//==================================================================================================
//							Beckhoff Automation Poland
//									23.05.2017
//	Program obslugujacy wizualizacje VISU_EventsHistoricalSimple
//	Mozliwe filtrowanie alamow. Czestotliwosc odswiezania wplywa tylko na wyswietlanie
// 	v1.0	|| TC v 3.1.4020.32		|| - pierwsza wersja
//==================================================================================================
PROGRAM P_EventsVisu
VAR
	i										: DINT;				// Iterator tablicy przechowywanej w pamieci
	j										: DINT;				// Iterator tablicy wyswietlanej
	bActiveWindow							: BOOL := TRUE;		// Flaga wysietlania okna - tylko wtedy odswiezamy tablice wyswietlana
	rtPageChange							: R_TRIG;			// Wykrycie przelaczenia strony
	tonRefresh								: TON;
	tRefreshTime							: TIME := T#50MS;	// Czestotliwosc odswiezania strony
	//========================= Filtry =========================
	bRemoveFromList							: BOOL; 			// Flaga pomocnicza dla filtrow - decyduje czy element ma byc dodany na wizualizacje
	// Flagi wykonywalnosci
	bFilterID								: BOOL;
	bFilterClass							: BOOL;
	bFilterActiveOnly						: BOOL;
	// Parametry
	dwFilterID								: DWORD;	
	dwFilterClass							: DWORD;
END_VAR

bActiveWindow := TRUE;//VisuElems.CURRENTVISU = 'VISU_EventsHistoricalSimple';						// Flaga wysietlania okna
rtPageChange(CLK:= bActiveWindow, Q=> );													// Wykrycie zmiany strony - jednorazowo inicjalizacja
tonRefresh(IN:= bActiveWindow AND NOT tonRefresh.Q, PT:= tRefreshTime, Q=> , ET=> );		// Timer odswiezania

IF  rtPageChange.Q OR tonRefresh.Q THEN
	// Czyszczenie tablicy
	MEMSET(ADR(GVL_EHS.arrEventVisu),0,SIZEOF(GVL_EHS.arrEventVisu));
	j := 1;
	// Filters
	FOR i := 1 TO GVL_EHS.diNoOfEvents DO
		bRemoveFromList 								:= FALSE;
		// Jesli jest element
		IF GVL_EHSP.arrEvent[i].dwID <> 0 THEN
			bRemoveFromList								:= bFilterID AND dwFilterID <> GVL_EHSP.arrEvent[i].dwID;
			bRemoveFromList								:= bRemoveFromList OR (bFilterClass AND dwFilterClass <> GVL_EHSP.arrEvent[i].dwClass);
//			bRemoveFromList								:= bRemoveFromList OR (bFilterBeginTimeFrom AND GVL_EHSP.arrEvent[i].dtDateBegin <= dtFilterBeginTimeFrom);
//			bRemoveFromList								:= bRemoveFromList OR (bFilterBeginTimeTo AND GVL_EHSP.arrEvent[i].dtDateBegin >= dtFilterBeginTimeTo);
//			bRemoveFromList								:= bRemoveFromList OR (bFilterEndTimeFrom AND GVL_EHSP.arrEvent[i].dtDateEnd <= dtFilterEndTimeFrom);
//			bRemoveFromList								:= bRemoveFromList OR (bFilterEndTimeTo AND GVL_EHSP.arrEvent[i].dtDateEnd >= dtFilterEndTimeTo);
			bRemoveFromList								:= bRemoveFromList OR (bFilterActiveOnly AND DT#1970-1-1-0:0:0 <> GVL_EHSP.arrEvent[i].dtDateEnd);
			// Analogicznie dodajemy inne filtry jesli jest taka potrzeba
			// Jesli element nie zostal usuniety przez filtr to dodajemy go do tablicy alarmow wyswietlanych
			IF NOT bRemoveFromList THEN
				GVL_EHS.arrEventVisu[j].dwID 			:= GVL_EHSP.arrEvent[i].dwID;
				GVL_EHS.arrEventVisu[j].dwClass 		:= GVL_EHSP.arrEvent[i].dwClass;
				GVL_EHS.arrEventVisu[j].wsMessage		:= GVL_EHS.arrEventDefinition[GVL_EHSP.arrEvent[i].dwID].wsMessage;
				GVL_EHS.arrEventVisu[j].dwParam 		:= GVL_EHSP.arrEvent[i].dwParam;
				GVL_EHS.arrEventVisu[j].dtDateBegin 	:= GVL_EHSP.arrEvent[i].dtDateBegin;
				GVL_EHS.arrEventVisu[j].dtDateEnd 		:= GVL_EHSP.arrEvent[i].dtDateEnd;
				IF GVL_EHS.arrEventVisu[j].dwClass=0 THEN
					GVL_EHS.arrEventVisu[j].dwColor:=16#FFFF0000;
				ELSIF GVL_EHS.arrEventVisu[j].dwClass=1 THEN
					GVL_EHS.arrEventVisu[j].dwColor:=16#FFF3F24A;
				ELSIF GVL_EHS.arrEventVisu[j].dwClass=2 THEN
					GVL_EHS.arrEventVisu[j].dwColor:=16#FF4E9640;
				END_IF
				j := j + 1;
			END_IF 
		END_IF
	END_FOR
END_IF

END_PROGRAM

(* stored: Version 1.1.0.1, ProductVersion 3.1.4022.7
   POU P_EventsVisu: Id {a09ad765-18f7-4e53-abc6-2a06babf9a29}, SpecialFunc None *)
